// TIA Portal V17 export
// export: Created 2021-12-03T08:12:55.5019871Z, ExportSetting WithDefaults, DisplayName Totally Integrated Automation Portal, DisplayVersion V17, DisplayName TIA Portal Openness, DisplayVersion V17, DisplayName TIA Portal Version Control Interface, DisplayVersion V17, DisplayName STEP 7 Professional, DisplayVersion V17, DisplayName STEP 7 Safety, DisplayVersion V17, DisplayName WinCC Advanced, DisplayVersion V17
DATA_BLOCK "DBI_DetLineCtrl"   // DB26
VERSION : 0.1
// stored: AutoNumber false, InstanceOfName FB_DetLineCtrl, InstanceOfType FB
"FB_DetLineCtrl"
   // VAR_INPUT
   //    ID : Int;
   //    LADDR : Word;
   //    I_StartScan : Bool;
   //    I_StopScan : Bool;
   //    I_Setup : Bool;
   //    I_Speed : Int;
   //    I_Direct : Bool;
   //    I_HighDose : Bool;
   // END_VAR
   // VAR RETAIN
   //    Telegr : Struct
   //       MsgID : DWord;
   //       MsgLen : DWord;
   //       ScanData : DWord;
   //       VehSpd : DWord;
   //    END_STRUCT;
   //    TCP_Sts : Struct
   //       Done : Bool;
   //       Error : Bool;
   //       Status : Word;
   //       Len : Int;
   //       ErrCd : Word;
   //    END_STRUCT;
   //    StrtTelegr : Bool;
   //    StrtTelegr_His : Bool;
   //    StrtTelegrSts : Bool;
   //    StrtTelegrSts_His : Bool;
   // END_VAR
BEGIN
END_DATA_BLOCK
